TYPE "RTrk_Item"
VERSION : 0.1
// Block: RTrk_Item
   STRUCT
      ID_R : DInt;
      PNo : DInt;
      WL_Indx : DInt;
      WL_Part : DInt;
      BeginPos : LReal;
      EndPos : LReal;
      Quality : Int;
   END_STRUCT;

END_TYPE
